TYPE ST_TransferMoldErrors :
STRUCT
	TrDidNotReachBMPosTimeOut		: BOOL;
	TrDidNotReachFormingPosTimeOut 	: BOOL;
	HydraulicCilinder				: ST_HydraulicErrorsAnalog;
END_STRUCT
END_TYPE

(* stored: Version 1.1.0.1, ProductVersion 3.1.4020.12
   DUT ST_TransferMoldErrors: Id {891babd8-6100-4e00-954e-204ae3c1dd7b} *)
